  rq_activate_all_grippers(False)
  # end: URCap Program Node
  $ 3 "Base_var≔Base_1_const"
  global Base_var=p[0.5798709432923697,-0.7737621037005363,-0.33271153235100037,-8.298354059056204E-4,0.017024779410152263,-3.136116651901569]
  $ 4 "Call Homee"
  Homee()
  # begin: URCap Program Node
  #   Source: OPC UA, 2.0.3, Rocketfarm AS
  #   Type: OPC UA Server
  $ 5 "Read OPC UA server: start"
  start =  opcua_server_read_byname("start")
  # end: URCap Program Node
  # begin: URCap Program Node
  #   Source: OPC UA, 2.0.3, Rocketfarm AS
  #   Type: OPC UA Server
  $ 6 "Read OPC UA server: isBusy"
  isBusy =  opcua_server_read_byname("isBusy")
  # end: URCap Program Node
  # begin: URCap Program Node
  #   Source: OPC UA, 2.0.3, Rocketfarm AS
  #   Type: OPC UA Server
  $ 7 "Read OPC UA server: service"
  service =  opcua_server_read_byname("service")
  # end: URCap Program Node
  # begin: URCap Program Node
  #   Source: OPC UA, 2.0.3, Rocketfarm AS
  #   Type: OPC UA Server
  $ 8 "Read OPC UA server: isUnderService"
  isUnderService =  opcua_server_read_byname("isUnderService")
  # end: URCap Program Node
  # begin: URCap Program Node
  #   Source: OPC UA, 2.0.3, Rocketfarm AS
  #   Type: OPC UA Server
  $ 9 "Read OPC UA server: pick_id"
  pick_id =  opcua_server_read_byname("pick_id")
  # end: URCap Program Node
  # begin: URCap Program Node
  #   Source: OPC UA, 2.0.3, Rocketfarm AS
  #   Type: OPC UA Server
  $ 10 "Read OPC UA server: pick_dir"
  pick_dir =  opcua_server_read_byname("pick_dir")
  # end: URCap Program Node
  # begin: URCap Program Node
  #   Source: OPC UA, 2.0.3, Rocketfarm AS
  #   Type: OPC UA Server
  $ 11 "Read OPC UA server: place_id"
  place_id =  opcua_server_read_byname("place_id")
  # end: URCap Program Node
  # begin: URCap Program Node
  #   Source: OPC UA, 2.0.3, Rocketfarm AS
  #   Type: OPC UA Server
  $ 12 "Read OPC UA server: place_dir"
  place_dir =  opcua_server_read_byname("place_dir")
  # end: URCap Program Node
  # begin: URCap Program Node
  #   Source: OPC UA, 2.0.3, Rocketfarm AS
  #   Type: OPC UA Server
  $ 13 "Read OPC UA server: atServicePosition"
  ServicePose =  opcua_server_read_byname("atServicePosition")
  # end: URCap Program Node
  while (True):
    $ 14 "Robot Program"
    $ 15 "Call Homee"
    Homee()
    $ 16 "Call openGripper"
    openGripper()
    $ 17 "Call Service"
    Service()
    $ 18 "Call wait_for_start"
    wait_for_start()
    $ 19 "Call read_pos"
    read_pos()
    $ 20 "Switch pick_dir"
    switch_1 = pick_dir
    $ 21 "Case 1"
    if (1 == switch_1):
      $ 22 "Base_var≔Base_1_const"
      global Base_var=p[0.5798709432923697,-0.7737621037005363,-0.33271153235100037,-8.298354059056204E-4,0.017024779410152263,-3.136116651901569]
    elif (2 == switch_1):
      $ 23 "Case 2"
      $ 24 "Base_var≔Base_2_const"
      global Base_var=p[-0.45890883940796207,-0.7057378570720949,-0.32683201510050314,0.005355978807793576,-0.00661010284054203,2.097302639945463]
    elif (3 == switch_1):
      $ 25 "Case 3"
      $ 26 "Base_var≔Base_3_const"
      global Base_var=p[-0.7619100891480977,0.45255476912365417,-0.31939996521398917,0.00889218721294195,0.00245126788755215,0.7004031128434923]
    elif (4 == switch_1):
      $ 27 "Case 4"
      $ 28 "Base_var≔Base_4_const"
      global Base_var=p[-0.7479251903865657,0.6881646623927705,-0.31636954411109924,-0.018501239315701457,0.007920304112792991,0.34091966894454795]
    elif (5 == switch_1):
      $ 29 "Case 5"
      $ 30 "Base_var≔Base_5_const"
      global Base_var=p[0.2190005627822054,1.00086979307141,-0.3124888627209852,0.02743720544787458,0.0036258560376326177,-0.7135956367863444]
    elif (6 == switch_1):
      $ 31 "Case 6"
      $ 32 "Base_var≔Base_6_const"
      global Base_var=p[0.9646176707982118,0.2060959762733794,-0.32472935894783184,0.00810684480276619,0.015634350758416675,-1.9383809628201483]
    else:
      $ 33 "Default Case"
      $ 34 "Halt"
      halt
    end
    $ 35 "Call Homee"
    Homee()
    $ 36 "Switch pick_id"
    switch_1 = pick_id
    $ 37 "Case 1"
    if (1 == switch_1):
      $ 38 "Call goPick_1"
      goPick_1()
    elif (2 == switch_1):
      $ 39 "Case 2"
      $ 40 "Call goPick_2"
      goPick_2()
    elif (101 == switch_1):
      $ 41 "Case 101"
      $ 42 "'test'"
      # 'test'
    else:
      $ 43 "Default Case"
      $ 44 "Halt"
      halt
    end
    $ 45 "Call Homee"
    Homee()
    $ 46 "Switch place_dir"
    switch_1 = place_dir
    $ 47 "Case 1"
    if (1 == switch_1):
      $ 48 "Base_var≔Base_1_const"
      global Base_var=p[0.5798709432923697,-0.7737621037005363,-0.33271153235100037,-8.298354059056204E-4,0.017024779410152263,-3.136116651901569]
    elif (2 == switch_1):
      $ 49 "Case 2"
      $ 50 "Base_var≔Base_2_const"
      global Base_var=p[-0.45890883940796207,-0.7057378570720949,-0.32683201510050314,0.005355978807793576,-0.00661010284054203,2.097302639945463]
    elif (3 == switch_1):
      $ 51 "Case 3"
      $ 52 "Base_var≔Base_3_const"
      global Base_var=p[-0.7619100891480977,0.45255476912365417,-0.31939996521398917,0.00889218721294195,0.00245126788755215,0.7004031128434923]
    elif (4 == switch_1):
      $ 53 "Case 4"
      $ 54 "Base_var≔Base_4_const"
      global Base_var=p[-0.7479251903865657,0.6881646623927705,-0.31636954411109924,-0.018501239315701457,0.007920304112792991,0.34091966894454795]
    elif (5 == switch_1):
      $ 55 "Case 5"
      $ 56 "Base_var≔Base_5_const"
      global Base_var=p[0.2190005627822054,1.00086979307141,-0.3124888627209852,0.02743720544787458,0.0036258560376326177,-0.7135956367863444]
    elif (6 == switch_1):
      $ 57 "Case 6"
      $ 58 "Base_var≔Base_6_const"
      global Base_var=p[0.9646176707982118,0.2060959762733794,-0.32472935894783184,0.00810684480276619,0.015634350758416675,-1.9383809628201483]
    else:
      $ 59 "Default Case"
      $ 60 "Halt"
      halt
    end
    $ 61 "Call Homee"
    Homee()
    $ 62 "Switch place_id"
    switch_1 = place_id
    $ 63 "Case 1"
    if (1 == switch_1):
      $ 64 "Call goPlace_1"
      goPlace_1()
    elif (2 == switch_1):
      $ 65 "Case 2"
      $ 66 "Call goPlace_2"
      goPlace_2()
    elif (101 == switch_1):
      $ 67 "Case 101"
      $ 68 "'test'"
      # 'test'
    else:
      $ 69 "Default Case"
      $ 70 "Halt"
      halt
    end
  end
end
